% RSLogix 500 project Practise-4.RSS, saved by version 8.30.00.16 %
PROJECT "UNTITLED"    % processor: MicroLogix 1000 %

PROGRAM FILES
  LAD 2 "MAIN_PROG"  6 rungs
  LAD 3 "USER_FAULT"  1 rungs
  LAD 4 "HSC_INT"  1 rungs
  LAD 5 "STI_INT"  1 rungs
  LAD 6, 7, 8, 9, 10, 11, 12, 13, 14, 15, 16: only END

DATA FILES
  O0 OUTPUT  1 elements
  I1 INPUT  2 elements
  S2 STATUS  33 elements
  B3 BINARY  32 elements
  T4 TIMER  40 elements
  C5 COUNTER  32 elements
  R6 CONTROL  16 elements
  N7 INTEGER  105 elements

LADDER 2 "MAIN_PROG"
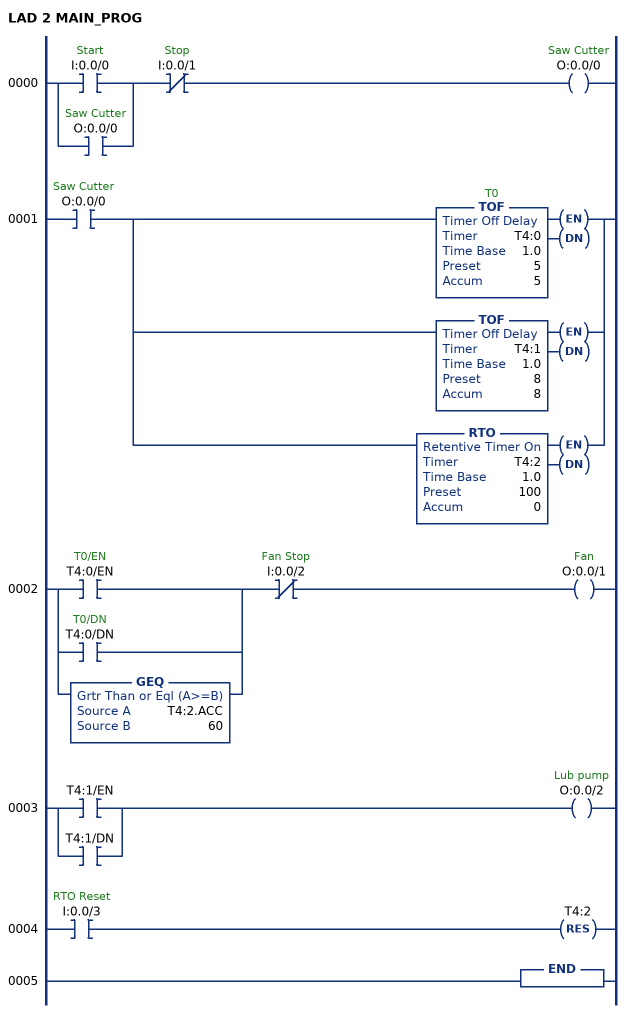
% Rung: 0 %
SOR BST XIC I:0.0/0 NXB XIC O:0.0/0 BND XIO I:0.0/1 OTE O:0.0/0 EOR
%   I:0.0/0  "Start" %
%   O:0.0/0  "Saw Cutter" %
%   I:0.0/1  "Stop" %
% Rung: 1 %
SOR XIC O:0.0/0 BST TOF T4:0 1.0 5 5 NXB BST TOF T4:1 1.0 8 8 NXB RTO T4:2 1.0 100 0 BND BND EOR
%   O:0.0/0  "Saw Cutter" %
%   T4:0  T0 %
% Rung: 2 %
SOR BST XIC T4:0/EN NXB BST XIC T4:0/DN NXB GEQ T4:2.ACC 60 BND BND XIO I:0.0/2 OTE O:0.0/1 EOR
%   T4:0  T0 %
%   I:0.0/2  "Fan Stop" %
%   O:0.0/1  "Fan" %
% Rung: 3 %
SOR BST XIC T4:1/EN NXB XIC T4:1/DN BND OTE O:0.0/2 EOR
%   O:0.0/2  "Lub pump" %
% Rung: 4 %
SOR XIC I:0.0/3 RES T4:2 EOR
%   I:0.0/3  "RTO Reset" %
% Rung: 5 %
SOR END EOR

DATA TABLE (non-zero values as saved)
DATA T4
% .PRE .ACC %
% T4:0 % 5 5
% T4:1 % 8 8
% T4:2 % 100 0
